TYPE "UDT_DeviceState"
TITLE = UDT_DeviceState
VERSION : 0.1
//User-defined structure of device states.
   STRUCT
      Configure { ExternalAccessible := 'False'; ExternalVisible := 'False'; ExternalWritable := 'False'} : Bool;   // Device configured in TIA Portal hardware
      Exist { ExternalAccessible := 'False'; ExternalVisible := 'False'; ExternalWritable := 'False'} : Bool;   // Device physically connected
      Error { ExternalAccessible := 'False'; ExternalVisible := 'False'; ExternalWritable := 'False'} : Bool;   // Device has an error
      ProfinetNumber : UInt;   // Profinet slave number
      HW_ID : UInt;   // Device's HW_ID
      PNDeviceName : String;   // Device's project name
   END_STRUCT;

END_TYPE

TYPE "UDT_ModuleState"
TITLE = UDT_ModuleState
VERSION : 0.1
//User-defined structure of module states.
   STRUCT
      Configured { ExternalAccessible := 'False'; ExternalVisible := 'False'; ExternalWritable := 'False'} : Bool;   // Module configured
      Exist { ExternalAccessible := 'False'; ExternalVisible := 'False'; ExternalWritable := 'False'} : Bool;   // Module exist
      Error { ExternalAccessible := 'False'; ExternalVisible := 'False'; ExternalWritable := 'False'} : Bool;   // Module has error
   END_STRUCT;

END_TYPE

TYPE "UDT_GINFedEx"
VERSION : 0.1
   STRUCT
      Timestamp : String[17];   // Local time timestamp
      TimeZoneDesignator : String[5];   // Time zone designator
      PackageEntrancePoint : String[14];   // Entrance point, where LLC starts tracking the parcel.
      PackageEntranceState : String[1];   // Entrance state
      PackageExitPoint : String[14];   // Exit point name, where LLC reports the last known tracking point.
      PackageExitState : String[1];   // Exit point state when LLC reports the last known tracking point.
      PalletType : String[2];   // Pallet code for different type of pallets on the market
      Mask : String[1];   // Flag to indicate that a pallet has been mask.
      CellNumber : String[4];   // Tray/Cell number (for loop sorters) or generated by LLC (on line sorters).
      CellsOccupied : String[1];   // Cells occupied by the piece for loop sorters.
      ImageID : String[6];   // Image ID number created by the ADC system.
      ScanUnitType : String[1];   // Scan unit type
      ADCSystemID : String[15];   // Number assigned by the ADC system
      PackageID : String[15];   // Number assigned by the LLC system
      LLCSystemID : String[15];
      HLCPackageID : String[10];   // Unique number for the specific package during it stays in HLC system.
      HLCResultCode : String[16];   // Result code based on processing of the scan event messages.
      ShipmentID : String[6];   // Consignment id of the parcel.
      WeightStatus : String[1];   // Status to indicate if the parcel/pallet has weight on the system.
      ActualDestination : String[6];   // Location code value that describes the actual disposition of the package.
      Destination1 : String[6];   // Location code value that describes where the package should go (Diverter Number).
      Destination2 : String[6];   // Location code value that describes where the package should go (Diverter Number).
      Destination3 : String[6];   // Location code value that describes where the package should go (Diverter Number).
      Destination4 : String[6];   // Location code value that describes where the package should go (Diverter Number).
      Destination5 : String[6];   // Location code value that describes where the package should go (Diverter Number).
      CutOffTimeDestination1 : String[5];   // Cut Off Time in Local Time.
      CutOffTimeDestination2 : String[5];   // Cut Off Time in Local Time.
      CutOffTimeDestination3 : String[5];   // Cut Off Time in Local Time.
      CutOffTimeDestination4 : String[5];   // Cut Off Time in Local Time.
      CutOffTimeDestination5 : String[5];   // Cut Off Time in Local Time.
      ReasonCode1 : String[8];   // Management Code value that describes the result of attempting to route the package to the Destination
      ReasonCode2 : String[8];   // Management Code value that describes the result of attempting to route the package to the Destination
      ReasonCode3 : String[8];   // Management Code value that describes the result of attempting to route the package to the Destination
      ReasonCode4 : String[8];   // Management Code value that describes the result of attempting to route the package to the Destination
      ReasonCode5 : String[8];   // Management Code value that describes the result of attempting to route the package to the Destination
      HLCDataText : String[20];   // Free text for future use.
      Customs : String[1];   // Need to be checked by customs
      DIMSystemID : String[15];   // Identifier of dimensioning system.
      DIMStatus : String[5];   // Basic diagnostic information from the dimensioning system at the moment of the measurement.
      PackageDimLength : String[6];   // Length dimension of package in resolution of dim system.
      PackageDimWidth : String[6];   // Width dimension of package in resolution of dim system.
      PackageDimHeight : String[6];   // Height dimension of package in resolution of dim system.
      DIMUOM : String[2];   // Unit of measure of the package dimensions.
      DimLFTstatusCode : String[8];   // Dimension LFT status code.
      DimConfidence : String[2];   // The level of assurance for the correct dimensions.
      DimensionSource : String[1];   // For combined camera/laser dim acquisition devices. It indicates type of capturing mode
      AlibiDims : String[25];   // Alibi for Dimensions
      SCLSystemID : String[15];   // Identifier of weight scale.
      SCLStatus : String[5];   // Basic diagnostic information from the weight scale system.
      SCLWT : String[6];   // Scale weight of package in resolution of scale system.
      SCLWTUOM : String[2];   // Unit of measurement for Weight
      SCLLFTStatusCode : String[2];   // Scale LFT status code.
      AlibiWeight : String[25];   // Alibi for Weight
      ReasonCode : String[1];   // This code should be used when the SI message has some defect.
      Stackable : String[1];   // If stackable recognition is enabled, Y or N
      Stickerstype : String[2];   // When optical recognition is used to sort
      FlyingDocument : String[1];   // Status to confirm if the document/flyer is prone to fly off the sorter.
      ModeofOperation : String[1];   // Camera Tunnel operational mode format:
      CameraHeadstatus : String[2];   // Diagnostic information on camera/laser heads performing barcode reads.
      PackageDataTruncated : String[1];   // Y = Full length of barcode data exceeds 9999 bytes, data truncated
      TotalBarcodeDataLength : String[4];   // Length of all barcode data that was sent in bytes;
      Barcode1Identification : String[3];   // Barcode identifier code.
      Barcode1status : String[2];   // Barcode confidence factor
      Barcode1datalength : String[4];   // String length of barcode data in bytes; inclusive of this field. Use 0054 as a fixed value
      Barcode1data : String[50];   // Highest priority barcode
      Barcode2Identification : String[3];   // Barcode identifier code.
      Barcode2status : String[2];   // Barcode confidence factor
      Barcode2datalength : String[4];   // String length of barcode data in bytes; inclusive of this field. Use 0054 as a fixed value
      Barcode2data : String[50];   // Highest priority barcode
      Barcode3Identification : String[3];   // Barcode identifier code.
      Barcode3status : String[2];   // Barcode confidence factor
      Barcode3datalength : String[4];   // String length of barcode data in bytes; inclusive of this field. Use 0054 as a fixed value
      Barcode3data : String[50];   // Highest priority barcode
      BarcodeIdentification : String[3];   // Barcode identifier code.
      Barcodestatus : String[2];   // Barcode confidence factor
      Barcodedatalength : String[4];   // String length of barcode data in bytes
      Barcodedata : String[50];   // Sortation barcode
      CustomerID : DInt;   // 6 digits SequentialID (NNNNNN)
      AreaNumber : String[2];   // Package Sequence ID "Area Number"
      PurgeEnabled { ExternalAccessible := 'False'; ExternalVisible := 'False'; ExternalWritable := 'False'} : Bool;   // Purge enabled for parcel: destination overwritten with Purge destination
   END_STRUCT;

END_TYPE

TYPE "UDT_GINStandard"
VERSION : 0.1
   STRUCT
      Destination : Array[0..20] of DInt;   // Destination
      Identification : Struct   // Barcode identification
         GoodRead { ExternalAccessible := 'False'; ExternalVisible := 'False'; ExternalWritable := 'False'} : Bool;   // Barcode read was succesful
         NoRead { ExternalAccessible := 'False'; ExternalVisible := 'False'; ExternalWritable := 'False'} : Bool;   // Barcode read was unsuccesful
         MultiRead { ExternalAccessible := 'False'; ExternalVisible := 'False'; ExternalWritable := 'False'} : Bool;   // Multiple Barcodes were detected
         Barcode : Array[0..10] of Char;   // Barcode values
      END_STRUCT;
      GinAssigned { ExternalAccessible := 'False'; ExternalVisible := 'False'; ExternalWritable := 'False'} : Bool;   // GIN is assigned to package
      Lost { ExternalAccessible := 'False'; ExternalVisible := 'False'; ExternalWritable := 'False'} : Bool;   // Lost in tracking
      Length : Int;   // Length in mm
      Width : Int;   // Width in mm
      Height : Int;   // Height in mm
      Weight : DInt;   // Weight in g
      PkgTooLong { ExternalAccessible := 'False'; ExternalVisible := 'False'; ExternalWritable := 'False'} : Bool;   // Package is too long
      PkgTooSmall { ExternalAccessible := 'False'; ExternalVisible := 'False'; ExternalWritable := 'False'} : Bool;   // Package is too small
      PkgTooHigh { ExternalAccessible := 'False'; ExternalVisible := 'False'; ExternalWritable := 'False'} : Bool;   // Package is too high
      PkgOverWeight { ExternalAccessible := 'False'; ExternalVisible := 'False'; ExternalWritable := 'False'} : Bool;   // Package is over weight
      TrailingGap : Int;   // Trailing gap size in cm between the package
      LeadingGap : Int;   // Leading gap size in cm between the package
      NrOfRecirculations : Int;   // Number of recirculations
      DestReqSend { ExternalAccessible := 'False'; ExternalVisible := 'False'; ExternalWritable := 'False'} : Bool;   // Destination request sent to high level
      DestRcv { ExternalAccessible := 'False'; ExternalVisible := 'False'; ExternalWritable := 'False'} : Bool;   // Destination received from high level
      SortStatus : Struct   // Sort status of the package
         DivertDestination : Int;   // Destination to which the package is diverted
         GoodDivert { ExternalAccessible := 'False'; ExternalVisible := 'False'; ExternalWritable := 'False'} : Bool;   // Package diverted
         FailedDivert { ExternalAccessible := 'False'; ExternalVisible := 'False'; ExternalWritable := 'False'} : Bool;   // Package failed to divert
         NoDivert : Bool := TRUE;   // Divert is not activated
         NoDivertCause : Struct   // Cause for no divert
            ChuteJam { ExternalAccessible := 'False'; ExternalVisible := 'False'; ExternalWritable := 'False'} : Bool;   // Chute is jammed
            ChuteFull { ExternalAccessible := 'False'; ExternalVisible := 'False'; ExternalWritable := 'False'} : Bool;   // Chute is full
            NoRTR { ExternalAccessible := 'False'; ExternalVisible := 'False'; ExternalWritable := 'False'} : Bool;   // Downstream conveyor is not ready to receive
            DestDisabled { ExternalAccessible := 'False'; ExternalVisible := 'False'; ExternalWritable := 'False'} : Bool;   // Destination is disabled
            TrayDisabled { ExternalAccessible := 'False'; ExternalVisible := 'False'; ExternalWritable := 'False'} : Bool;   // Tray is disabled
            SorterNotAtSpeed { ExternalAccessible := 'False'; ExternalVisible := 'False'; ExternalWritable := 'False'} : Bool;   // Sorter is not at speed
            LeadingGapError { ExternalAccessible := 'False'; ExternalVisible := 'False'; ExternalWritable := 'False'} : Bool;   // Gap size with downstream parcel is not enough
            TrailingGapError { ExternalAccessible := 'False'; ExternalVisible := 'False'; ExternalWritable := 'False'} : Bool;   // Gap size with upstream parcel is not enough
            PkgTooHigh { ExternalAccessible := 'False'; ExternalVisible := 'False'; ExternalWritable := 'False'} : Bool;   // Package is too high to divert
            PkgTooLong { ExternalAccessible := 'False'; ExternalVisible := 'False'; ExternalWritable := 'False'} : Bool;   // Package is too long to divert
            DestNotReachable { ExternalAccessible := 'False'; ExternalVisible := 'False'; ExternalWritable := 'False'} : Bool;   // Sort destionation is not reachable
            InvalidDest { ExternalAccessible := 'False'; ExternalVisible := 'False'; ExternalWritable := 'False'} : Bool;   // Sort destination is invalid
            DestTooLate { ExternalAccessible := 'False'; ExternalVisible := 'False'; ExternalWritable := 'False'} : Bool;   // Destination too late
            NoDestRcv { ExternalAccessible := 'False'; ExternalVisible := 'False'; ExternalWritable := 'False'} : Bool;   // Destination not received from high level
         END_STRUCT;
      END_STRUCT;
   END_STRUCT;

END_TYPE

TYPE "UDT_GINWES"
VERSION : 0.1
   STRUCT
      Barcode : String[40];
   END_STRUCT;

END_TYPE

TYPE "UDT_GINWCS"
VERSION : 0.1
   STRUCT
      ActionTaken : String;   // Location code value that describes the actual disposition of the package
      Destination1 : String[20];   // Location code value that describes where the package should go (Diverter Number)
      Destination2 : String[20];   // Location code value that describes where the package should go (Diverter Number)
      Destination3 : String[20];   // Location code value that describes where the package should go (Diverter Number)
      Destination4 : String[20];   // Location code value that describes where the package should go (Diverter Number)
      Destination5 : String[20];   // Location code value that describes where the package should go (Diverter Number)
      ReasonCode : String[2];   // Management Code value that describes the result of attempting to route the package to the Destination
      Barcode1 : String;   // Barcode identifier code
      Barcode2 : String;
      Barcode3 : String;
      Barcode4 : String;
   END_STRUCT;

END_TYPE

TYPE "UDT_GINDHL"
VERSION : 0.1
   STRUCT
      ObjectID : String[10];   // Object ID
      VID : String[16];   // Virtual Item Identifier (VID)
      PieceID : String[40];   // Piece ID barcodes
      SortStrategy : String[1];   // Sort Strategy 1 - Highest priority available , 2 - Nearest
      ParcelReject { ExternalAccessible := 'False'; ExternalVisible := 'False'; ExternalWritable := 'False'} : Bool;   // True - Parcel reject
      Destination : Array[1..6] of Struct   // Destination
         ID : UInt;   // ID
         SortCommandActive { ExternalAccessible := 'False'; ExternalVisible := 'False'; ExternalWritable := 'False'} : Bool;   // Sort command
         ParcelSorted { ExternalAccessible := 'False'; ExternalVisible := 'False'; ExternalWritable := 'False'} : Bool;   // Parcel sorted
         Rejected { ExternalAccessible := 'False'; ExternalVisible := 'False'; ExternalWritable := 'False'} : Bool;   // Parcel rejected
         Reason : Int;   // Reason
      END_STRUCT;
      ParcelLocation : Struct   // Parcel Location
         Current : UInt;   // Current
         Last : UInt;   // Last
         Sort : UInt;   // Sort
      END_STRUCT;
      MFCMessage : Struct   // MFC Sort messages
         Sent : Struct   // Messages sent from the PLC to the MFC system
            SortResult { ExternalAccessible := 'False'; ExternalVisible := 'False'; ExternalWritable := 'False'} : Bool;   // Message Sort Result
            VIDResponse { ExternalAccessible := 'False'; ExternalVisible := 'False'; ExternalWritable := 'False'} : Bool;   // Message VID Response
            ScanReset { ExternalAccessible := 'False'; ExternalVisible := 'False'; ExternalWritable := 'False'} : Bool;   // Message Scan Reset
            XrayResult { ExternalAccessible := 'False'; ExternalVisible := 'False'; ExternalWritable := 'False'} : Bool;   // Message Xray result
            ParcelRegInfo { ExternalAccessible := 'False'; ExternalVisible := 'False'; ExternalWritable := 'False'} : Bool;   // Message Xray registration info
         END_STRUCT;
         Received : Struct   // Messages received from the MFC system to the PLC
            RejectParcel { ExternalAccessible := 'False'; ExternalVisible := 'False'; ExternalWritable := 'False'} : Bool;   // Message Reject Parcel
            Destination { ExternalAccessible := 'False'; ExternalVisible := 'False'; ExternalWritable := 'False'} : Bool;   // Message Destination
            DestinationResent { ExternalAccessible := 'False'; ExternalVisible := 'False'; ExternalWritable := 'False'} : Bool;   // Message Destination Resent
            TemporaryParcelIdentifier { ExternalAccessible := 'False'; ExternalVisible := 'False'; ExternalWritable := 'False'} : Bool;   // Message Temporary Parcel Identifier
            XrayRegistrationInfo { ExternalAccessible := 'False'; ExternalVisible := 'False'; ExternalWritable := 'False'} : Bool;
         END_STRUCT;
      END_STRUCT;
      Xray : Struct   // Xray data structure
         RoutingCode : String[2];   // Routing code
         Group : String[1];   // The group field is used to identify the group of the operator decisions came from in a
         Level : String[1];   // Level field is used to identify which level the operator decision came from in a
         Result : String[1];   // Results can be indicated with the following:A = Accept, R = Reject, U = Unavailable (Timeout), Z = High Threat
         BagIDMessage : Struct   // Message from PLC to Xray
            MessagePrepared { ExternalAccessible := 'False'; ExternalVisible := 'False'; ExternalWritable := 'False'} : Bool;   // The message is prepared and ready to send
            WrongMessageStructure { ExternalAccessible := 'False'; ExternalVisible := 'False'; ExternalWritable := 'False'} : Bool;   // The message has wrong structure
            Sent { ExternalAccessible := 'False'; ExternalVisible := 'False'; ExternalWritable := 'False'} : Bool;   // The message sent by PLC to Xray
            SentTime : String;   // Time when message sent by PLC to Xray
            NotSent { ExternalAccessible := 'False'; ExternalVisible := 'False'; ExternalWritable := 'False'} : Bool;   // The message was not sent from the PLC
            Received { ExternalAccessible := 'False'; ExternalVisible := 'False'; ExternalWritable := 'False'} : Bool;   // The message received by Xray
            TimeReceived : String;   // Time when message received by Xray
            NotReceived { ExternalAccessible := 'False'; ExternalVisible := 'False'; ExternalWritable := 'False'} : Bool;   // The message did not reach Xray
         END_STRUCT;
         DecisionMessage : Struct   // Message from Xray to PLC
            Received { ExternalAccessible := 'False'; ExternalVisible := 'False'; ExternalWritable := 'False'} : Bool;   // The message received by PLC
            ReceivedTime : String;   // The message received by PLC
            NotReceivedOnTime { ExternalAccessible := 'False'; ExternalVisible := 'False'; ExternalWritable := 'False'} : Bool;   // The message did not reach PLC
         END_STRUCT;
      END_STRUCT;
   END_STRUCT;

END_TYPE

TYPE "UDT_CommonStatus"
TITLE = UDT_CommonStatus
VERSION : 0.1
//User-defined structure of common statuses.
   STRUCT
      SafetyStop { ExternalAccessible := 'False'; ExternalVisible := 'False'; ExternalWritable := 'False'} : Bool;   // Emergancy stop
      Error { ExternalAccessible := 'False'; ExternalVisible := 'False'; ExternalWritable := 'False'} : Bool;   // An error is active
      Warning { ExternalAccessible := 'False'; ExternalVisible := 'False'; ExternalWritable := 'False'} : Bool;   // A warning is active
      ManualRun { ExternalAccessible := 'False'; ExternalVisible := 'False'; ExternalWritable := 'False'} : Bool;   // Running in manual mode
      Manual { ExternalAccessible := 'False'; ExternalVisible := 'False'; ExternalWritable := 'False'} : Bool;   // In manual mode
      Halted { ExternalAccessible := 'False'; ExternalVisible := 'False'; ExternalWritable := 'False'} : Bool;   // Halted
      Dieback { ExternalAccessible := 'False'; ExternalVisible := 'False'; ExternalWritable := 'False'} : Bool;   // In dieback
      Stopped { ExternalAccessible := 'False'; ExternalVisible := 'False'; ExternalWritable := 'False'} : Bool;   // Stopped
      Running { ExternalAccessible := 'False'; ExternalVisible := 'False'; ExternalWritable := 'False'} : Bool;   // Running
      EnergySave { ExternalAccessible := 'False'; ExternalVisible := 'False'; ExternalWritable := 'False'} : Bool;   // In energy saving mode
      AutoON { ExternalAccessible := 'False'; ExternalVisible := 'False'; ExternalWritable := 'False'} : Bool;   // Automatic started
   END_STRUCT;

END_TYPE

TYPE "UDT_EventStatistic"
TITLE = UDT_EventStatistic
VERSION : 0.1
//User-defined structure of event statistic data.
   STRUCT
      NumberOfTimes : DInt;   // Number of times the event occurred since last reset
      LastEventSeconds : DInt;   // Number of seconds of the current or last event
      TotalEventSeconds : DInt;   // Total number of seconds the event occurred since last reset
   END_STRUCT;

END_TYPE

TYPE "UDT_GINUPS"
VERSION : 0.1
   STRUCT
      TRKNUM : String[18];   // Tracking number
      PKGUID : String[32];   // Package ID
      MSGID : String[32];   // Message ID
      Length : Int;   // Camera Length in mm
      Width : Int;   // Camera Width in mm
      Height : Int;   // Camera Height in mm
      Weight : DInt;   // Weight in g
      IDCreated { ExternalAccessible := 'False'; ExternalVisible := 'False'; ExternalWritable := 'False'} : Bool;   // Byte 1, Bit 0 - PLCID created or TrayID Read
      DimDataRcv { ExternalAccessible := 'False'; ExternalVisible := 'False'; ExternalWritable := 'False'} : Bool;   // Byte 1, Bit 1 - Package Dimensional Data Received via Camera Scan Data Message
      PkgWrongInduct { ExternalAccessible := 'False'; ExternalVisible := 'False'; ExternalWritable := 'False'} : Bool;   // Byte 1, Bit 2 - Package Did NOT Induct Properly (Non-Tray Systems)
      IDCalcFromCamID { ExternalAccessible := 'False'; ExternalVisible := 'False'; ExternalWritable := 'False'} : Bool;   // Byte 2, Bit 0 - PLCID/TrayID Calculated From CamID
      UnknownParcelID { ExternalAccessible := 'False'; ExternalVisible := 'False'; ExternalWritable := 'False'} : Bool;   // Byte 2, Bit 4 - Unknown Parcel ID
      UndefinedProblem { ExternalAccessible := 'False'; ExternalVisible := 'False'; ExternalWritable := 'False'} : Bool;   // Byte 2, Bit 5 - Un-Defined Problem
      UnrecognizedCmd { ExternalAccessible := 'False'; ExternalVisible := 'False'; ExternalWritable := 'False'} : Bool;   // Byte 2, Bit 6 - Un-recognized command
      SorterInMainteneceMode { ExternalAccessible := 'False'; ExternalVisible := 'False'; ExternalWritable := 'False'} : Bool;   // Byte 2, Bit 7 - Sorter in Maintenance/Commissioning Mode
      DestUserSusp { ExternalAccessible := 'False'; ExternalVisible := 'False'; ExternalWritable := 'False'} : Bool;   // Byte 3, Bit 3 - Destination User Suspended
      SorterNotSynch { ExternalAccessible := 'False'; ExternalVisible := 'False'; ExternalWritable := 'False'} : Bool;   // Byte 3, Bit 6 - Sorter NOT Synchronized (Tilt Tray Systems)
      PkgDetAtVerCheckPoint { ExternalAccessible := 'False'; ExternalVisible := 'False'; ExternalWritable := 'False'} : Bool;   // Byte 4, Bit 0 - Package Detected at Verification Check Point
      ChuteFullAftrAlterDest { ExternalAccessible := 'False'; ExternalVisible := 'False'; ExternalWritable := 'False'} : Bool;   // Byte 4, Bit 7 - Preferred chute full after passed alternate destination
      ChuteNotAvailAfterAlterDest { ExternalAccessible := 'False'; ExternalVisible := 'False'; ExternalWritable := 'False'} : Bool;   // Byte 5, Bit 0 - Preferred chute not available after passed alternate destination
      PLCRedirected { ExternalAccessible := 'False'; ExternalVisible := 'False'; ExternalWritable := 'False'} : Bool;   // Byte 5, Bit 2 - PLC Redirected
      ThreatParcel { ExternalAccessible := 'False'; ExternalVisible := 'False'; ExternalWritable := 'False'} : Bool;   // Threat parcel
   END_STRUCT;

END_TYPE

TYPE "UDT_ProfinetDevice"
TITLE = UDT_ProfinetDevice
VERSION : 0.1
//User-defined structure of profinet device state.
   STRUCT
      DeviceState : "UDT_DeviceState";   // Device state
      Module { S7_SetPoint := 'False'} : Array[0..31] of "UDT_ModuleState";   // Modules
   END_STRUCT;

END_TYPE

TYPE "UDT_Message"
TITLE = UDT_Message
VERSION : 0.1
//User-defined structure of the message characters array.
   STRUCT
      Character : Array[0..499] of Char;   // Message character
   END_STRUCT;

END_TYPE

TYPE "UDT_FifoHeader"
TITLE = UDT_FifoHeader
VERSION : 0.1
//User-defined structure of FIFO register header information.
   STRUCT
      Status : Struct   // Status bits
         Empty { ExternalAccessible := 'False'; ExternalVisible := 'False'; ExternalWritable := 'False'} : Bool;   // FIFO Empty
         Prefull { ExternalAccessible := 'False'; ExternalVisible := 'False'; ExternalWritable := 'False'} : Bool;   // FIFO Prefull
         Full { ExternalAccessible := 'False'; ExternalVisible := 'False'; ExternalWritable := 'False'} : Bool;   // FIFO Full
      END_STRUCT;
      NextEntryToRead : Int;   // Next FIFO entry to read
      NextEntryToWrite : Int;   // Next FIFO entry to write
      MaxNrOfEntries : Int;   // Maximum number of FIFO entries
      TotalEntriesStored : Int;   // Total number of FIFO entries
   END_STRUCT;

END_TYPE

TYPE "UDT_ProfiDiagStatistics"
TITLE = UDT_ProfiDiagStatistics
VERSION : 0.1
//User-defined structure of FB_ProfiDiag function block statistics.
   STRUCT
      DeviceError { S7_SetPoint := 'False'} : Array[0..512] of "UDT_EventStatistic";   // Device error statistics
   END_STRUCT;

END_TYPE

TYPE "UDT_Connection"
TITLE = UDT_Connection
VERSION : 0.1
//User-defined structure of connection parameters.
   STRUCT
      ActiveEstablished : Bool := FALSE;   // 0 – Passive connection establishment; 1 – Active connection establishment
      Interface_ID : HW_ANY := 64;   // Interface ID of CPU Ethernet interface
      ID : CONN_OUC;   // Unique ID as system reference for the connection
      IP : Array[1..4] of Int;   // IP address
      Port : UInt;   // Port number of the communication partner
      ConTimeout : DInt;   // Maximum waiting time for response from the communication partner [ms]
   END_STRUCT;

END_TYPE

TYPE "UDT_PowerDistributionPanelCBState"
VERSION : 0.1
   STRUCT
      CircuitBreakerStateF100 { ExternalAccessible := 'False'; ExternalVisible := 'False'; ExternalWritable := 'False'} : Bool;   // Circuit Breaker State Ok if the signal is true
      CircuitBreakerStateF201 { ExternalAccessible := 'False'; ExternalVisible := 'False'; ExternalWritable := 'False'} : Bool;   // Circuit Breaker State Ok if the signal is true
      CircuitBreakerStateF202 { ExternalAccessible := 'False'; ExternalVisible := 'False'; ExternalWritable := 'False'} : Bool;   // Circuit Breaker State Ok if the signal is true
      CircuitBreakerStateF203 { ExternalAccessible := 'False'; ExternalVisible := 'False'; ExternalWritable := 'False'} : Bool;   // Circuit Breaker State Ok if the signal is true
      CircuitBreakerStateF204 { ExternalAccessible := 'False'; ExternalVisible := 'False'; ExternalWritable := 'False'} : Bool;   // Circuit Breaker State Ok if the signal is true
      CircuitBreakerStateF205 { ExternalAccessible := 'False'; ExternalVisible := 'False'; ExternalWritable := 'False'} : Bool;   // Circuit Breaker State Ok if the signal is true
      CircuitBreakerStateF206 { ExternalAccessible := 'False'; ExternalVisible := 'False'; ExternalWritable := 'False'} : Bool;   // Circuit Breaker State Ok if the signal is true
      CircuitBreakerStateF207 { ExternalAccessible := 'False'; ExternalVisible := 'False'; ExternalWritable := 'False'} : Bool;   // Circuit Breaker State Ok if the signal is true
      CircuitBreakerStateF208 { ExternalAccessible := 'False'; ExternalVisible := 'False'; ExternalWritable := 'False'} : Bool;   // Circuit Breaker State Ok if the signal is true
      CircuitBreakerStateF209 { ExternalAccessible := 'False'; ExternalVisible := 'False'; ExternalWritable := 'False'} : Bool;   // Circuit Breaker State Ok if the signal is true
      CircuitBreakerStateF210 { ExternalAccessible := 'False'; ExternalVisible := 'False'; ExternalWritable := 'False'} : Bool;   // Circuit Breaker State Ok if the signal is true
      CircuitBreakerStateF211 { ExternalAccessible := 'False'; ExternalVisible := 'False'; ExternalWritable := 'False'} : Bool;   // Circuit Breaker State Ok if the signal is true
      CircuitBreakerStateF212 { ExternalAccessible := 'False'; ExternalVisible := 'False'; ExternalWritable := 'False'} : Bool;   // Circuit Breaker State Ok if the signal is true
      CircuitBreakerStateF213 { ExternalAccessible := 'False'; ExternalVisible := 'False'; ExternalWritable := 'False'} : Bool;   // Circuit Breaker State Ok if the signal is true
      CircuitBreakerStateF214 { ExternalAccessible := 'False'; ExternalVisible := 'False'; ExternalWritable := 'False'} : Bool;   // Circuit Breaker State Ok if the signal is true
      CircuitBreakerStateF215 { ExternalAccessible := 'False'; ExternalVisible := 'False'; ExternalWritable := 'False'} : Bool;   // Circuit Breaker State Ok if the signal is true
      CircuitBreakerStateF216 { ExternalAccessible := 'False'; ExternalVisible := 'False'; ExternalWritable := 'False'} : Bool;   // Circuit Breaker State Ok if the signal is true
      CircuitBreakerStateF217 { ExternalAccessible := 'False'; ExternalVisible := 'False'; ExternalWritable := 'False'} : Bool;   // Circuit Breaker State Ok if the signal is true
      CircuitBreakerStateF218 { ExternalAccessible := 'False'; ExternalVisible := 'False'; ExternalWritable := 'False'} : Bool;   // Circuit Breaker State Ok if the signal is true
      CircuitBreakerStateF219 { ExternalAccessible := 'False'; ExternalVisible := 'False'; ExternalWritable := 'False'} : Bool;   // Circuit Breaker State Ok if the signal is true
      CircuitBreakerStateF220 { ExternalAccessible := 'False'; ExternalVisible := 'False'; ExternalWritable := 'False'} : Bool;   // Circuit Breaker State Ok if the signal is true
      CircuitBreakerStateF221 { ExternalAccessible := 'False'; ExternalVisible := 'False'; ExternalWritable := 'False'} : Bool;   // Circuit Breaker State Ok if the signal is true
      CircuitBreakerStateF222 { ExternalAccessible := 'False'; ExternalVisible := 'False'; ExternalWritable := 'False'} : Bool;   // Circuit Breaker State Ok if the signal is true
      CircuitBreakerStateF223 { ExternalAccessible := 'False'; ExternalVisible := 'False'; ExternalWritable := 'False'} : Bool;   // Circuit Breaker State Ok if the signal is true
      CircuitBreakerStateF224 { ExternalAccessible := 'False'; ExternalVisible := 'False'; ExternalWritable := 'False'} : Bool;   // Circuit Breaker State Ok if the signal is true
      CircuitBreakerStateF225 { ExternalAccessible := 'False'; ExternalVisible := 'False'; ExternalWritable := 'False'} : Bool;   // Circuit Breaker State Ok if the signal is true
      CircuitBreakerStateF226 { ExternalAccessible := 'False'; ExternalVisible := 'False'; ExternalWritable := 'False'} : Bool;   // Circuit Breaker State Ok if the signal is true
      CircuitBreakerStateF227 { ExternalAccessible := 'False'; ExternalVisible := 'False'; ExternalWritable := 'False'} : Bool;   // Circuit Breaker State Ok if the signal is true
      CircuitBreakerStateF228 { ExternalAccessible := 'False'; ExternalVisible := 'False'; ExternalWritable := 'False'} : Bool;   // Circuit Breaker State Ok if the signal is true
      CircuitBreakerStateF229 { ExternalAccessible := 'False'; ExternalVisible := 'False'; ExternalWritable := 'False'} : Bool;   // Circuit Breaker State Ok if the signal is true
      CircuitBreakerStateF230 { ExternalAccessible := 'False'; ExternalVisible := 'False'; ExternalWritable := 'False'} : Bool;   // Circuit Breaker State Ok if the signal is true
      CircuitBreakerStateF231 { ExternalAccessible := 'False'; ExternalVisible := 'False'; ExternalWritable := 'False'} : Bool;   // Circuit Breaker State Ok if the signal is true
      CircuitBreakerStateF232 { ExternalAccessible := 'False'; ExternalVisible := 'False'; ExternalWritable := 'False'} : Bool;   // Circuit Breaker State Ok if the signal is true
      CircuitBreakerStateF233 { ExternalAccessible := 'False'; ExternalVisible := 'False'; ExternalWritable := 'False'} : Bool;   // Circuit Breaker State Ok if the signal is true
      CircuitBreakerStateF234 { ExternalAccessible := 'False'; ExternalVisible := 'False'; ExternalWritable := 'False'} : Bool;   // Circuit Breaker State Ok if the signal is true
      CircuitBreakerStateF235 { ExternalAccessible := 'False'; ExternalVisible := 'False'; ExternalWritable := 'False'} : Bool;   // Circuit Breaker State Ok if the signal is true
      CircuitBreakerStateF236 { ExternalAccessible := 'False'; ExternalVisible := 'False'; ExternalWritable := 'False'} : Bool;   // Circuit Breaker State Ok if the signal is true
      CircuitBreakerStateF237 { ExternalAccessible := 'False'; ExternalVisible := 'False'; ExternalWritable := 'False'} : Bool;   // Circuit Breaker State Ok if the signal is true
      CircuitBreakerStateF238 { ExternalAccessible := 'False'; ExternalVisible := 'False'; ExternalWritable := 'False'} : Bool;   // Circuit Breaker State Ok if the signal is true
      CircuitBreakerStateF239 { ExternalAccessible := 'False'; ExternalVisible := 'False'; ExternalWritable := 'False'} : Bool;   // Circuit Breaker State Ok if the signal is true
      CircuitBreakerStateF240 { ExternalAccessible := 'False'; ExternalVisible := 'False'; ExternalWritable := 'False'} : Bool;   // Circuit Breaker State Ok if the signal is true
      CircuitBreakerStateF241 { ExternalAccessible := 'False'; ExternalVisible := 'False'; ExternalWritable := 'False'} : Bool;   // Circuit Breaker State Ok if the signal is true
      CircuitBreakerStateF242 { ExternalAccessible := 'False'; ExternalVisible := 'False'; ExternalWritable := 'False'} : Bool;   // Circuit Breaker State Ok if the signal is true
      CircuitBreakerStateF243 { ExternalAccessible := 'False'; ExternalVisible := 'False'; ExternalWritable := 'False'} : Bool;   // Circuit Breaker State Ok if the signal is true
      CircuitBreakerStateF244 { ExternalAccessible := 'False'; ExternalVisible := 'False'; ExternalWritable := 'False'} : Bool;   // Circuit Breaker State Ok if the signal is true
      CircuitBreakerStateF245 { ExternalAccessible := 'False'; ExternalVisible := 'False'; ExternalWritable := 'False'} : Bool;   // Circuit Breaker State Ok if the signal is true
      CircuitBreakerStateF246 { ExternalAccessible := 'False'; ExternalVisible := 'False'; ExternalWritable := 'False'} : Bool;   // Circuit Breaker State Ok if the signal is true
      CircuitBreakerStateF247 { ExternalAccessible := 'False'; ExternalVisible := 'False'; ExternalWritable := 'False'} : Bool;   // Circuit Breaker State Ok if the signal is true
      CircuitBreakerStateF248 { ExternalAccessible := 'False'; ExternalVisible := 'False'; ExternalWritable := 'False'} : Bool;   // Circuit Breaker State Ok if the signal is true
      CircuitBreakerStateF249 { ExternalAccessible := 'False'; ExternalVisible := 'False'; ExternalWritable := 'False'} : Bool;   // Circuit Breaker State Ok if the signal is true
      CircuitBreakerStateF250 { ExternalAccessible := 'False'; ExternalVisible := 'False'; ExternalWritable := 'False'} : Bool;   // Circuit Breaker State Ok if the signal is true
      CircuitBreakerStateF251 { ExternalAccessible := 'False'; ExternalVisible := 'False'; ExternalWritable := 'False'} : Bool;   // Circuit Breaker State Ok if the signal is true
      CircuitBreakerStateF501 { ExternalAccessible := 'False'; ExternalVisible := 'False'; ExternalWritable := 'False'} : Bool;   // Circuit Breaker State Ok if the signal is true
      CircuitBreakerStateF502 { ExternalAccessible := 'False'; ExternalVisible := 'False'; ExternalWritable := 'False'} : Bool;   // Circuit Breaker State Ok if the signal is true
      CircuitBreakerStateF503 { ExternalAccessible := 'False'; ExternalVisible := 'False'; ExternalWritable := 'False'} : Bool;   // Circuit Breaker State Ok if the signal is true
      CircuitBreakerStateF504 { ExternalAccessible := 'False'; ExternalVisible := 'False'; ExternalWritable := 'False'} : Bool;   // Circuit Breaker State Ok if the signal is true
      CircuitBreakerStateF505 { ExternalAccessible := 'False'; ExternalVisible := 'False'; ExternalWritable := 'False'} : Bool;   // Circuit Breaker State Ok if the signal is true
   END_STRUCT;

END_TYPE

TYPE "UDT_EquipmentControl"
TITLE = UDT_EquipmentControl
VERSION : 0.1
//User-defined structure of equipment control commands.
   STRUCT
      Command : Struct   // Control command
         Start { ExternalAccessible := 'False'; ExternalVisible := 'False'; ExternalWritable := 'False'} : Bool;   // Start conveyor
         Stop { ExternalAccessible := 'False'; ExternalVisible := 'False'; ExternalWritable := 'False'} : Bool;   // Stop conveyor
         Reset { ExternalAccessible := 'False'; ExternalVisible := 'False'; ExternalWritable := 'False'} : Bool;   // Faults reset
         ResetData { ExternalAccessible := 'False'; ExternalVisible := 'False'; ExternalWritable := 'False'} : Bool;   // Statistics reset
         ManualMode { ExternalAccessible := 'False'; ExternalVisible := 'False'; ExternalWritable := 'False'} : Bool;   // Manual mode required
         DisableManualMode { ExternalAccessible := 'False'; ExternalVisible := 'False'; ExternalWritable := 'False'} : Bool;   // Disable manual mode
         AutomaticOn { ExternalAccessible := 'False'; ExternalVisible := 'False'; ExternalWritable := 'False'} : Bool;   // System is started in automatic mode
         StopRequest { ExternalAccessible := 'False'; ExternalVisible := 'False'; ExternalWritable := 'False'} : Bool;
      END_STRUCT;
      Report { S7_SetPoint := 'False'} : "UDT_CommonStatus";   // Conveyors state
      Request : Struct   // Request from equipment
         RestartRequired { ExternalAccessible := 'False'; ExternalVisible := 'False'; ExternalWritable := 'False'} : Bool;   // Restart required from system control
         SignalingRequest { ExternalAccessible := 'False'; ExternalVisible := 'False'; ExternalWritable := 'False'} : Bool;   // Beeper required
         InhibitStop { ExternalAccessible := 'False'; ExternalVisible := 'False'; ExternalWritable := 'False'} : Bool;
      END_STRUCT;
   END_STRUCT;

END_TYPE

TYPE "UDT_ProfinetNetwork"
TITLE = UDT_ProfinetNetwork
VERSION : 0.1
//User-defined structure of profinet network state.
   STRUCT
      DeviceStatus : Array[0..512] of "UDT_ProfinetDevice";   // Profinet device status
   END_STRUCT;

END_TYPE

TYPE "UDT_ControlPowerGroupStatistics"
VERSION : 0.1
   STRUCT
      PowerSupplyGroupWarnning : "UDT_EventStatistic";   // Warning Power Supply Group Statistics
      PowerSupplyGroupError : "UDT_EventStatistic";   // Error Power Supply Group Statistics
   END_STRUCT;

END_TYPE

TYPE "UDT_TCPIPConnectStatistics"
TITLE = UDT_TCPIPConnectStatistics
VERSION : 0.1
//User-defined structure of FB_TCPIPConnect function block statistics.
   STRUCT
      ConnectionLost { S7_SetPoint := 'False'} : "UDT_EventStatistic";   // Connection lost statistics
   END_STRUCT;

END_TYPE

TYPE "UDT_TCPIPReceiveStatistics"
TITLE = UDT_TCPIPReceiveStatistics
VERSION : 0.1
//User-defined structure of FB_TCPIPReceive function block statistics.
   STRUCT
      InvalidMsg : UInt;   // Invalid message received
   END_STRUCT;

END_TYPE

TYPE "UDT_WSRBufferState"
VERSION : 0.1
   STRUCT
      Destination : Int;
      BufferState1 : Struct
         BinRequest : Bool;
         BinSend : Bool;
         UpcomingBarcode : String[30];
         WaintingTime : Int;
      END_STRUCT;
      BufferState2 : Struct
         BinRequest : Bool;
         BinSend : Bool;
         UpcomingBarcode : String[30];
         WaintingTime : Int;
      END_STRUCT;
      BufferState3 : Struct
         BinRequest : Bool;
         BinSend : Bool;
         UpcomingBarcode : String[30];
         WaintingTime : Int;
      END_STRUCT;
   END_STRUCT;

END_TYPE

TYPE "UDT_SystemControlStatus"
TITLE = UDT_SystemControlStatus
VERSION : 0.1
//User-defined structure of FB_SystemControl function block status.
   STRUCT
      Status : Int;   // Status number
   END_STRUCT;

END_TYPE

TYPE "UDT_ControlPowerGroupStatus"
VERSION : 0.1
   STRUCT
      Status : Int;   // Status number
      Specific : Struct
         Fail_PowerSupply_1 { ExternalAccessible := 'False'; ExternalVisible := 'False'; ExternalWritable := 'False'} : Bool;   // Power supply 1 fail
         Fail_PowerSupply_2 { ExternalAccessible := 'False'; ExternalVisible := 'False'; ExternalWritable := 'False'} : Bool;   // Power supply 2 fail
         Fail_PowerSupply_3 { ExternalAccessible := 'False'; ExternalVisible := 'False'; ExternalWritable := 'False'} : Bool;   // Power supply 3 fail
         Fail_PowerSupply_4 { ExternalAccessible := 'False'; ExternalVisible := 'False'; ExternalWritable := 'False'} : Bool;   // Power supply 4 fail
         Fail_PowerSupply_5 { ExternalAccessible := 'False'; ExternalVisible := 'False'; ExternalWritable := 'False'} : Bool;   // Power supply 5 fail
         Fail_PowerSupply_6 { ExternalAccessible := 'False'; ExternalVisible := 'False'; ExternalWritable := 'False'} : Bool;   // Power supply 6 fail
         Fail_PowerSupply_7 { ExternalAccessible := 'False'; ExternalVisible := 'False'; ExternalWritable := 'False'} : Bool;   // Power supply 7 fail
         Fail_PowerSupply_8 { ExternalAccessible := 'False'; ExternalVisible := 'False'; ExternalWritable := 'False'} : Bool;   // Power supply 8 fail
         Fail_PowerSupply_9 { ExternalAccessible := 'False'; ExternalVisible := 'False'; ExternalWritable := 'False'} : Bool;   // Power supply 9 fail
         Fail_PowerSupply_10 { ExternalAccessible := 'False'; ExternalVisible := 'False'; ExternalWritable := 'False'} : Bool;   // Power supply 10 fail
         PowerSuppliesWarning { ExternalAccessible := 'False'; ExternalVisible := 'False'; ExternalWritable := 'False'} : Bool;   // Power supplies warning
         PowerSuppliesError { ExternalAccessible := 'False'; ExternalVisible := 'False'; ExternalWritable := 'False'} : Bool;   // Power supplies error
      END_STRUCT;
   END_STRUCT;

END_TYPE

TYPE "UDT_MainControlPanelStatus"
TITLE = Cabinet MCP Status
VERSION : 0.1
   STRUCT
      Status : Int;   //  Status number
      Specific : Struct
         PN_PN_MSP_PNSlaveNotOnline { ExternalAccessible := 'False'; ExternalVisible := 'False'; ExternalWritable := 'False'} : Bool;   //  PNPN coupler is not online
         PN_PN_MSP_PNSlaveError { ExternalAccessible := 'False'; ExternalVisible := 'False'; ExternalWritable := 'False'} : Bool;   //  PNPN coupler has an error
         PN_PN_MSP_PNSlaveWarning { ExternalAccessible := 'False'; ExternalVisible := 'False'; ExternalWritable := 'False'} : Bool;   //  PNPN coupler has a warning
         IOModule_PNSlaveNotOnline { ExternalAccessible := 'False'; ExternalVisible := 'False'; ExternalWritable := 'False'} : Bool;   // I/O Module is not online
         IOModule_PNSlaveError { ExternalAccessible := 'False'; ExternalVisible := 'False'; ExternalWritable := 'False'} : Bool;   // I/O Module has an error
         IOModule_PNSlaveWarning { ExternalAccessible := 'False'; ExternalVisible := 'False'; ExternalWritable := 'False'} : Bool;   // I/O Module has a warning
         ScalanceSwitchPNSlaveNotOnline { ExternalAccessible := 'False'; ExternalVisible := 'False'; ExternalWritable := 'False'} : Bool;   // Scalance switch is not online
         ScalanceSwitchPNSlaveError { ExternalAccessible := 'False'; ExternalVisible := 'False'; ExternalWritable := 'False'} : Bool;   // Scalance switch has an error
         ScalanceSwitchPNSlaveWarning { ExternalAccessible := 'False'; ExternalVisible := 'False'; ExternalWritable := 'False'} : Bool;   // Scalance switch has a warning
         ScalanceSwitchStatus { ExternalAccessible := 'False'; ExternalVisible := 'False'; ExternalWritable := 'False'} : Bool;   // TRUE when Scalance switch is not healthy
         Singulator_PNSlaveNotOnline { ExternalAccessible := 'False'; ExternalVisible := 'False'; ExternalWritable := 'False'} : Bool;   // Singulator coupler is not online
         Singulator_PNSlaveError { ExternalAccessible := 'False'; ExternalVisible := 'False'; ExternalWritable := 'False'} : Bool;   // Singulator coupler has an error
         Singulator_PNSlaveWarning { ExternalAccessible := 'False'; ExternalVisible := 'False'; ExternalWritable := 'False'} : Bool;   // Singulator coupler has a warning
         UPSSwitchTripped { ExternalAccessible := 'False'; ExternalVisible := 'False'; ExternalWritable := 'False'} : Bool;   //  Unit Power Supply switch tripped
         FireAlarmActive { ExternalAccessible := 'False'; ExternalVisible := 'False'; ExternalWritable := 'False'} : Bool;   //  Fire alarm active when the signal is true
         PS_201T1_Tripped { ExternalAccessible := 'False'; ExternalVisible := 'False'; ExternalWritable := 'False'} : Bool;   //  TRUE if power supply 201T1 tripped
         "230VAC_CB201F4Tripped" { ExternalAccessible := 'False'; ExternalVisible := 'False'; ExternalWritable := 'False'} : Bool;   //  TRUE if MCP circuit breaker 201F4 tripped
         "230VAC_CB101F1Tripped" { ExternalAccessible := 'False'; ExternalVisible := 'False'; ExternalWritable := 'False'} : Bool;   //  TRUE if MCP circuit breaker 101F1 tripped
         "230VAC_CB101F4Tripped" { ExternalAccessible := 'False'; ExternalVisible := 'False'; ExternalWritable := 'False'} : Bool;   //  TRUE if MCP circuit breaker 101F4 tripped
         "230VAC_CB102F1Tripped" { ExternalAccessible := 'False'; ExternalVisible := 'False'; ExternalWritable := 'False'} : Bool;   //  TRUE if MCU circuit breaker 102F1 tripped
         "230VAC_CB102F3Tripped" { ExternalAccessible := 'False'; ExternalVisible := 'False'; ExternalWritable := 'False'} : Bool;   //  TRUE if MCU circuit breaker 102F3 tripped
         "24VDC_CB201F1Tripped" { ExternalAccessible := 'False'; ExternalVisible := 'False'; ExternalWritable := 'False'} : Bool;   //  TRUE if MCU circuit breaker 205F1 tripped
         "24VDC_CB205F5Tripped" { ExternalAccessible := 'False'; ExternalVisible := 'False'; ExternalWritable := 'False'} : Bool;   //  TRUE if MCU circuit breaker 205F5 tripped
         "24VDC_CB205F9Tripped" { ExternalAccessible := 'False'; ExternalVisible := 'False'; ExternalWritable := 'False'} : Bool;   //  TRUE if MCU circuit breaker 205F9 tripped
         Spare_1 { ExternalAccessible := 'False'; ExternalVisible := 'False'; ExternalWritable := 'False'} : Bool;   // Spare
         Spare_2 { ExternalAccessible := 'False'; ExternalVisible := 'False'; ExternalWritable := 'False'} : Bool;   // Spare
         Spare_3 { ExternalAccessible := 'False'; ExternalVisible := 'False'; ExternalWritable := 'False'} : Bool;   // Spare
         RackSlotError : Array[0..31] of Bool;   //  One of the main rack slots has an error
         IOModuleSlotError : Array[0..31] of Bool;   //  Module error
      END_STRUCT;
   END_STRUCT;

END_TYPE

TYPE "UDT_TCPIPConnectStatus"
TITLE = UDT_TCPIPConnectStatus
VERSION : 0.1
//User-defined structure of FB_TCPIPConnect function block status.
   STRUCT
      Status : Int;   // Status number
      Specific : Struct   // Specific status structure
         ErrorCode : Struct   // Error code structure
            TCON : Word;   // Siemens TCON error code - Check documetation
            TDISCON : Word;   // Siemens TDISCON error code - Check documetation
            TDIAG : Word;   // Siemens TDIAG error code - Check documetation
         END_STRUCT;
         Connected { ExternalAccessible := 'False'; ExternalVisible := 'False'; ExternalWritable := 'False'} : Bool;   // Connected
         CommunicationFault { ExternalAccessible := 'False'; ExternalVisible := 'False'; ExternalWritable := 'False'} : Bool;   // Communication fault
      END_STRUCT;
   END_STRUCT;

END_TYPE

TYPE "UDT_UnknownGIN"
TITLE = UDT_UnknownGIN
VERSION : 0.1
//User-defined structure of unknown GIN range.
   STRUCT
      Start : Int := 1;   // Unknown GIN range start value
      End : Int := 199;   // Unknown GIN range end value
      GIN : Int := 0;   // Las generated unknown GIN
   END_STRUCT;

END_TYPE

TYPE "UDT_GOSLog"
VERSION : 0.1
   STRUCT
      GIN_nr : Int;
      InfeedUpstreamGap : Int;   // Gap in millimeters (mm)
      InfeedDownstreamGap : Int;   // Gap in millimeters (mm)
      OutfeedUpstreamGap : Int;   // Gap in meters (mm)
      OutfeedDownstreamGap : Int;   // Gap in meters (mm)
      ParcelLength : Int;
      GapToBeRecovered : Int;
      ParcelDownStreamResults : Int;
      ParcelUpStreamResults : Int;
      Accelerate { ExternalAccessible := 'False'; ExternalVisible := 'False'; ExternalWritable := 'False'} : Bool;
      Decelerate { ExternalAccessible := 'False'; ExternalVisible := 'False'; ExternalWritable := 'False'} : Bool;
      PrevConveyorUpstreamGap : Int;
      PrevConveyorDownstreamGap : Int;
      NextConveyorUpstreamGap : Int;
      NextConveyorDownstreamGap : Int;
   END_STRUCT;

END_TYPE

TYPE "UDT_GIN"
VERSION : 0.1
   STRUCT
      General { S7_SetPoint := 'False'} : "UDT_GINStandard";
      FedEx { S7_SetPoint := 'False'} : "UDT_GINFedEx";
      UPS { S7_SetPoint := 'False'} : "UDT_GINUPS";
      DHL { S7_SetPoint := 'False'} : "UDT_GINDHL";
      WCS { S7_SetPoint := 'False'} : "UDT_GINWCS";
      WES { S7_SetPoint := 'False'} : "UDT_GINWES";
   END_STRUCT;

END_TYPE

TYPE "UDT_MainControlPanelStatistics"
TITLE = Cabinet MCP Statistics
VERSION : 0.1
   STRUCT
      UPSFault : "UDT_EventStatistic";   // Unit Power Supply fault statistics
      FireAlarm : "UDT_EventStatistic";   // Fire Alarm active statistics
      "230VAC_CB101F1Tripped" : "UDT_EventStatistic";   // Circuit braker 101F1 tripped  statistics
      "230VAC_CB101F4Tripped" : "UDT_EventStatistic";   // Circuit braker 101F4 tripped statistics
      "230VAC_CB102F1Tripped" : "UDT_EventStatistic";   // Circuit braker 102F1 tripped statistics
      "230VAC_CB102F3Tripped" : "UDT_EventStatistic";   // Circuit braker 102F3 tripped statistics
      "230VAC_CB201F4Tripped" : "UDT_EventStatistic";   // Circuit braker 201F4 tripped statistics
      "24VDC_CB201F1Tripped" : "UDT_EventStatistic";   // Circuit braker 201F1 tripped statistics
      "24VDC_CB205F5Tripped" : "UDT_EventStatistic";   // Circuit braker 205F5 tripped statistics
      "24VDC_CB205F9Tripped" : "UDT_EventStatistic";   // Circuit braker 205F9 tripped statistics
      ScalanceSwitchStatus : "UDT_EventStatistic";   // Scalance switch status statistics
      Spare_1 : "UDT_EventStatistic";   // Spare
      Spare_2 : "UDT_EventStatistic";   // Spare
      Spare_3 : "UDT_EventStatistic";   // Spare
      PS_201T1_Tripped { S7_SetPoint := 'False'} : "UDT_EventStatistic";   // Circuit braker 201T1 tripped statistics
      "PN/PNCouplerFault" : "UDT_EventStatistic";   // PN/PN coupler fault statistics
      SingulatorCouplerFault : "UDT_EventStatistic";   // ProSoft coupler fault statistics
      ScalanceSwitchFault : "UDT_EventStatistic";   // Scalance switch fault statistics
      IOModuleCouplerFault : "UDT_EventStatistic";   // IO Module fault statistics
      RackModuleFault : "UDT_EventStatistic";   // A module fault occurred in the mainrack
   END_STRUCT;

END_TYPE

TYPE "UDT_SystemControlCommand"
TITLE = UDT_SystemControlCommand
VERSION : 0.1
//User-defined structure of system control commands.
   STRUCT
      Start { ExternalAccessible := 'False'; ExternalVisible := 'False'; ExternalWritable := 'False'} : Bool;   // Start Command from HMI
      Stop { ExternalAccessible := 'False'; ExternalVisible := 'False'; ExternalWritable := 'False'} : Bool;   // Stop command from HMI
      Reset { ExternalAccessible := 'False'; ExternalVisible := 'False'; ExternalWritable := 'False'} : Bool;   // Reset command from HMI
      ResetData { ExternalAccessible := 'False'; ExternalVisible := 'False'; ExternalWritable := 'False'} : Bool;   // Reset data command from HMI
      ResetSafety { ExternalAccessible := 'False'; ExternalVisible := 'False'; ExternalWritable := 'False'} : Bool;   // Reset safety command from HMI
      ManualMode { ExternalAccessible := 'False'; ExternalVisible := 'False'; ExternalWritable := 'False'} : Bool;   // Manual mode command from HMI
   END_STRUCT;

END_TYPE

DATA_BLOCK "DB_FIFOMedPrioMsg"
TITLE = DB_FIFO
{ S7_Optimized_Access := 'TRUE' }
AUTHOR : MHSE
FAMILY : GeneralSystemFunctions
VERSION : 3.0
NON_RETAIN
//Data block to store FIFO registers.
   VAR RETAIN
      Header { ExternalAccessible := 'False'; ExternalVisible := 'False'; ExternalWritable := 'False'; S7_SetPoint := 'False'} : "UDT_FifoHeader";   // FIFO Header
      Data { ExternalAccessible := 'False'; ExternalVisible := 'False'; ExternalWritable := 'False'; S7_SetPoint := 'False'} : Array[0..199] of "UDT_Message";   // FIFO data buffer
   END_VAR


BEGIN

END_DATA_BLOCK

DATA_BLOCK "DB_FIFORcvMsg"
TITLE = DB_FIFO
{ S7_Optimized_Access := 'TRUE' }
AUTHOR : MHSE
FAMILY : GeneralSystemFunctions
VERSION : 3.0
NON_RETAIN
//Data block to store FIFO registers.
   VAR RETAIN
      Header { ExternalAccessible := 'False'; ExternalVisible := 'False'; ExternalWritable := 'False'; S7_SetPoint := 'False'} : "UDT_FifoHeader";   // FIFO Header
      Data { ExternalAccessible := 'False'; ExternalVisible := 'False'; ExternalWritable := 'False'; S7_SetPoint := 'False'} : Array[0..199] of "UDT_Message";   // FIFO data buffer
   END_VAR


BEGIN

END_DATA_BLOCK

DATA_BLOCK "DB_Configuration"
TITLE = DB_Configuration
{ S7_Optimized_Access := 'TRUE' }
AUTHOR : MHSE
FAMILY : GeneralSystemFunctions
VERSION : 3.0
NON_RETAIN
//Data block to store configuration data.
   VAR RETAIN
      System { ExternalAccessible := 'False'; ExternalVisible := 'False'; ExternalWritable := 'False'} : Struct   // System configuration
         Connection { ExternalAccessible := 'False'; ExternalVisible := 'False'; ExternalWritable := 'False'} : "UDT_Connection";   // Connection configuration
      END_STRUCT;
   END_VAR


BEGIN
   System.Connection.ActiveEstablished := TRUE;
   System.Connection.Interface_ID := 64;
   System.Connection.ID := 16#0001;
   System.Connection.IP[1] := 192;
   System.Connection.IP[2] := 168;
   System.Connection.IP[3] := 3;
   System.Connection.IP[4] := 53;
   System.Connection.Port := 42300;
   System.Connection.ConTimeout := 5000;

END_DATA_BLOCK

DATA_BLOCK "DB_FIFOHighPrioMsg"
TITLE = DB_FIFO
{ S7_Optimized_Access := 'TRUE' }
AUTHOR : MHSE
FAMILY : GeneralSystemFunctions
VERSION : 3.0
NON_RETAIN
//Data block to store FIFO registers.
   VAR
      Header { ExternalAccessible := 'False'; ExternalVisible := 'False'; ExternalWritable := 'False'; S7_SetPoint := 'False'} : "UDT_FifoHeader";   // FIFO Header
      Data { ExternalAccessible := 'False'; ExternalVisible := 'False'; ExternalWritable := 'False'; S7_SetPoint := 'False'} : Array[0..199] of "UDT_Message";   // FIFO data buffer
   END_VAR


BEGIN

END_DATA_BLOCK

DATA_BLOCK "DB_ExternalHandshake"
TITLE = DB_ExternalHandshake
{ S7_Optimized_Access := 'TRUE' }
AUTHOR : MHSE
FAMILY : Equimpent
VERSION : 3.0
NON_RETAIN
//Data block to store external equipment handshake data.

BEGIN

END_DATA_BLOCK

DATA_BLOCK "DB_Control"
{ S7_Optimized_Access := 'TRUE' }
AUTHOR : MHSE
FAMILY : Equimpent
VERSION : 0.1
NON_RETAIN
   VAR
      System1 { ExternalAccessible := 'False'; ExternalVisible := 'False'; ExternalWritable := 'False'; S7_SetPoint := 'False'} : "UDT_EquipmentControl";
   END_VAR


BEGIN

END_DATA_BLOCK

DATA_BLOCK "DB_Communication"
TITLE = DB_Communication
{ S7_Optimized_Access := 'TRUE' }
AUTHOR : MHSE
FAMILY : Communication
VERSION : 3.0
NON_RETAIN
//Data block to store communication data.
   VAR
      BuildingMnemonic { ExternalAccessible := 'False'; ExternalVisible := 'False'; ExternalWritable := 'False'} : String[5];   // Building mnemonic
      ModuleName { ExternalAccessible := 'False'; ExternalVisible := 'False'; ExternalWritable := 'False'} : String[2];   // Module type
      DeviceNumber { ExternalAccessible := 'False'; ExternalVisible := 'False'; ExternalWritable := 'False'} : String[4];   // Device number
   END_VAR


BEGIN
   BuildingMnemonic := 'abcde';
   ModuleName := 'AB';
   DeviceNumber := 'abcd';

END_DATA_BLOCK

DATA_BLOCK "DB_WSRManager"
{ S7_Optimized_Access := 'TRUE' }
VERSION : 0.1
NON_RETAIN
   VAR
      EmptyFifoHeader { ExternalAccessible := 'False'; ExternalVisible := 'False'; ExternalWritable := 'False'; S7_SetPoint := 'False'} : "UDT_FifoHeader";
      EmptyFifoData { ExternalAccessible := 'False'; ExternalVisible := 'False'; ExternalWritable := 'False'} : Array[0..110] of Int;
      PartialFifoHeader { ExternalAccessible := 'False'; ExternalVisible := 'False'; ExternalWritable := 'False'; S7_SetPoint := 'False'} : "UDT_FifoHeader";
      PartialFifoData { ExternalAccessible := 'False'; ExternalVisible := 'False'; ExternalWritable := 'False'} : Array[0..110] of Int;
      WSR01Empty { ExternalAccessible := 'False'; ExternalVisible := 'False'; ExternalWritable := 'False'; S7_SetPoint := 'False'} : Array[0..18] of "UDT_WSRBufferState";
      WSR01Partial { ExternalAccessible := 'False'; ExternalVisible := 'False'; ExternalWritable := 'False'; S7_SetPoint := 'False'} : Array[0..18] of "UDT_WSRBufferState";
   END_VAR


BEGIN

END_DATA_BLOCK

DATA_BLOCK "DB_RATPositioning"
{ S7_Optimized_Access := 'TRUE' }
VERSION : 0.1
NON_RETAIN

BEGIN

END_DATA_BLOCK

DATA_BLOCK "DB_GOSLog"
{ S7_Optimized_Access := 'TRUE' }
VERSION : 0.1
NON_RETAIN
   VAR
      DB_GOSLog { ExternalAccessible := 'False'; ExternalVisible := 'False'; ExternalWritable := 'False'; S7_SetPoint := 'False'} : Array[0..100] of "UDT_GOSLog";
   END_VAR


BEGIN

END_DATA_BLOCK

DATA_BLOCK "DB_ExternalGIN"
{ S7_Optimized_Access := 'TRUE' }
VERSION : 0.1
NON_RETAIN
   VAR
      UnexpectedSI { ExternalAccessible := 'False'; ExternalVisible := 'False'; ExternalWritable := 'False'; S7_SetPoint := 'False'} : "UDT_GIN";
   END_VAR


BEGIN

END_DATA_BLOCK

DATA_BLOCK "DB_HMISpeed"
{ S7_Optimized_Access := 'TRUE' }
VERSION : 0.1
NON_RETAIN
   VAR
      Dummy : Int;
   END_VAR


BEGIN

END_DATA_BLOCK

DATA_BLOCK "DB_Variables"
{ S7_Optimized_Access := 'TRUE' }
VERSION : 0.1
NON_RETAIN
   VAR
      CIP_StopRequest { ExternalAccessible := 'False'; ExternalVisible := 'False'; ExternalWritable := 'False'} : Bool;   // System stop request from CIP
      ResetEnergySave { ExternalAccessible := 'False'; ExternalVisible := 'False'; ExternalWritable := 'False'} : Bool;   // When True Reset Energy Save mode
      StartToSystemControl { ExternalAccessible := 'False'; ExternalVisible := 'False'; ExternalWritable := 'False'} : Bool;   // From SSP Lamp to System Control
      ResetToSystemControl { ExternalAccessible := 'False'; ExternalVisible := 'False'; ExternalWritable := 'False'} : Bool;   // From SSP Lamp to System Control
   END_VAR


BEGIN

END_DATA_BLOCK

DATA_BLOCK "DB_FIFOLowPrioMsg"
TITLE = DB_FIFO
{ S7_Optimized_Access := 'TRUE' }
AUTHOR : MHSE
FAMILY : GeneralSystemFunctions
VERSION : 3.0
NON_RETAIN
//Data block to store FIFO registers.
   VAR RETAIN
      Header { ExternalAccessible := 'False'; ExternalVisible := 'False'; ExternalWritable := 'False'; S7_SetPoint := 'False'} : "UDT_FifoHeader";   // FIFO Header
      Data { ExternalAccessible := 'False'; ExternalVisible := 'False'; ExternalWritable := 'False'; S7_SetPoint := 'False'} : Array[0..199] of "UDT_Message";   // FIFO data buffer
   END_VAR


BEGIN

END_DATA_BLOCK

DATA_BLOCK "DB_ProgrammingError"
{ S7_Optimized_Access := 'TRUE' }
VERSION : 0.1
NON_RETAIN
   VAR
      NrOfErrors { ExternalAccessible := 'False'; ExternalVisible := 'False'; ExternalWritable := 'False'} : Int;
      BlockNr { ExternalAccessible := 'False'; ExternalVisible := 'False'; ExternalWritable := 'False'} : UInt;
      Reaction { ExternalAccessible := 'False'; ExternalVisible := 'False'; ExternalWritable := 'False'} : USInt;
      Fault_ID { ExternalAccessible := 'False'; ExternalVisible := 'False'; ExternalWritable := 'False'} : Byte;
      BlockType { ExternalAccessible := 'False'; ExternalVisible := 'False'; ExternalWritable := 'False'} : USInt;
      Area { ExternalAccessible := 'False'; ExternalVisible := 'False'; ExternalWritable := 'False'} : USInt;
      DBNr { ExternalAccessible := 'False'; ExternalVisible := 'False'; ExternalWritable := 'False'} : DB_ANY;
      Csg_OBNr { ExternalAccessible := 'False'; ExternalVisible := 'False'; ExternalWritable := 'False'} : OB_ANY;
      Csg_Prio { ExternalAccessible := 'False'; ExternalVisible := 'False'; ExternalWritable := 'False'} : USInt;
      Width { ExternalAccessible := 'False'; ExternalVisible := 'False'; ExternalWritable := 'False'} : USInt;
   END_VAR


BEGIN

END_DATA_BLOCK

DATA_BLOCK "DB_HMIStatusConfiguration"
TITLE = DB_HMIStatusConfiguration
{ S7_Optimized_Access := 'TRUE' }
AUTHOR : MHSE
VERSION : 3.0
NON_RETAIN
   VAR
      FireAlarm : Int;   // Fire alarm active
      SafetyStop : Int;   // Safety stop error status
      Error : Int;   // Error status
      Warning : Int;   // Warning status
      ManualRun : Int;   // Manual run status
      Manual : Int;   // Manual status
      Halted : Int;   // Halted status
      Dieback : Int;   // Die back status
      Stopped : Int;   // Stopped status
      Running : Int;   // Running status
      EnergySave : Int;   // Energy save status
      CommunicationError : Int;   // Communication error status
      CBError : Int;   // CB error status
      ProfinetError : Int;   // Profinet error status
      HardwareError : Int;   // Hardware error status
      VFDNotHealthy : Int;   // VFD noth healthy status
      VFDError : Int;   // VFD error status
      PECJam : Int;   // PEC jam status
      ChuteFull : Int;   // Chute full status
      EncoderError : Int;   // Encoder error status
      TrackingError : Int;   // Tracking error status
      DimensionError : Int;   // Dimension error status
      OperationalError : Int;   // Operational error status
      AutoON : Int;   // Automatic is on
      ChuteHalfFull : Int;   // Disable by operator
      DisableByManagement : Int;   // Disable by management
      GateOpen : Int;   // Manual operated gate is open
      GateClosed : Int;   // Manual operated gate is closed
      GateClosedAndNoOperatorPresent : Int;   // Manual operated gate is closed and no operator is present
      PositionChangeOngoing : Int;   // Lifting device or arm diverter changing position
      BufferMode : Int;   // BufferMode Active
      ContinuousMode : Int;   // ContinuousMode Active
      LabbelingMode : Int;   // LabbelingMode Active
   END_VAR


BEGIN
   FireAlarm := 1;
   SafetyStop := 3;
   Error := 5;
   Warning := 7;
   ManualRun := 9;
   Manual := 11;
   Halted := 13;
   Dieback := 15;
   Stopped := 17;
   Running := 19;
   EnergySave := 21;
   CommunicationError := 23;
   CBError := 25;
   ProfinetError := 27;
   HardwareError := 29;
   VFDNotHealthy := 31;
   VFDError := 33;
   PECJam := 35;
   ChuteFull := 37;
   EncoderError := 39;
   TrackingError := 41;
   DimensionError := 43;
   OperationalError := 45;
   AutoON := 47;
   ChuteHalfFull := 49;
   DisableByManagement := 51;
   GateOpen := 53;
   GateClosed := 55;
   GateClosedAndNoOperatorPresent := 57;
   PositionChangeOngoing := 59;
   BufferMode := 61;
   ContinuousMode := 63;
   LabbelingMode := 65;

END_DATA_BLOCK

DATA_BLOCK "DB_Handshake"
TITLE = DB_Handshake
{ S7_Optimized_Access := 'TRUE' }
AUTHOR : MHSE
FAMILY : Equimpent
VERSION : 3.0
NON_RETAIN
//Data block to store equipment handshake data.

BEGIN

END_DATA_BLOCK

DATA_BLOCK "DB_SafetyInterface"
{ S7_Optimized_Access := 'TRUE' }
VERSION : 0.1
NON_RETAIN
   VAR
      SafetyReset { ExternalAccessible := 'False'; ExternalVisible := 'False'; ExternalWritable := 'False'} : Bool;
   END_VAR


BEGIN

END_DATA_BLOCK

DATA_BLOCK "DB_MotorData"
{ S7_Optimized_Access := 'TRUE' }
VERSION : 0.1
NON_RETAIN

BEGIN

END_DATA_BLOCK

DATA_BLOCK "DB_VFDCommissioningControl"
{ S7_Optimized_Access := 'TRUE' }
VERSION : 0.1
NON_RETAIN
   VAR
      dummy_Start { ExternalAccessible := 'False'; ExternalVisible := 'False'; ExternalWritable := 'False'} : Bool;   // start VFD Commissioning
      dummy_GoToNextStep { ExternalAccessible := 'False'; ExternalVisible := 'False'; ExternalWritable := 'False'} : Bool;   // Trigger to move into the next step
   END_VAR


BEGIN

END_DATA_BLOCK

DATA_BLOCK "DB_HardwareOK"
{ S7_Optimized_Access := 'TRUE' }
VERSION : 0.1
NON_RETAIN
   VAR
      System { ExternalAccessible := 'False'; ExternalVisible := 'False'; ExternalWritable := 'False'} : Struct   // System status
         MCP { ExternalAccessible := 'False'; ExternalVisible := 'False'; ExternalWritable := 'False'} : Bool;   // Main Control Panel
         CPG01 { ExternalAccessible := 'False'; ExternalVisible := 'False'; ExternalWritable := 'False'} : Bool;
      END_STRUCT;
   END_VAR


BEGIN

END_DATA_BLOCK

DATA_BLOCK "DB_CommonStatus"
TITLE = DB_Status
{ S7_Optimized_Access := 'TRUE' }
AUTHOR : MHSE
FAMILY : GeneralSystemFunctions
VERSION : 3.0
NON_RETAIN
//Data block to store status data.
   VAR
      Communication : Struct   // Communication status
         TCPIPConnect : "UDT_CommonStatus";   // FB_TCPIPConnect status
      END_STRUCT;
      System : Struct   // System statuses
         System1 { S7_SetPoint := 'False'} : "UDT_CommonStatus";
         MCP { S7_SetPoint := 'False'} : "UDT_CommonStatus";
         CPG01 : "UDT_CommonStatus";
         CPG02 : "UDT_CommonStatus";
         CPG03 : "UDT_CommonStatus";
         CPG04 : "UDT_CommonStatus";
         CPG05 : "UDT_CommonStatus";
         test { S7_SetPoint := 'True'} : Int;
      END_STRUCT;
   END_VAR


BEGIN

END_DATA_BLOCK

DATA_BLOCK "DB_UnknownGINRange"
TITLE = DB_UnknownGINRange
{ S7_Optimized_Access := 'TRUE' }
AUTHOR : MHSE
FAMILY : GeneralSystemFunctions
VERSION : 3.0
NON_RETAIN
//Data block to store unknown GIN range data.
   VAR RETAIN
      UnknownGINRange { ExternalAccessible := 'False'; ExternalVisible := 'False'; ExternalWritable := 'False'; S7_SetPoint := 'False'} : "UDT_UnknownGIN";   // Unknown GIN range structure
   END_VAR


BEGIN

END_DATA_BLOCK

DATA_BLOCK "DB_Time"
TITLE = DB_Time
{ S7_Optimized_Access := 'TRUE' }
AUTHOR : MHSE
FAMILY : GeneralSystemFunctions
VERSION : 3.0
NON_RETAIN
//Data block to store date and time data.
   VAR
      ActualTimeDTL {InstructionName := 'DTL'; LibVersion := '1.0'; ExternalAccessible := 'False'; ExternalVisible := 'False'; ExternalWritable := 'False'} : DTL;   // Actual date and time in DTL
      ActualTime { ExternalAccessible := 'False'; ExternalVisible := 'False'; ExternalWritable := 'False'} : String;   // Actual date and time in String
      Timestamp { ExternalAccessible := 'False'; ExternalVisible := 'False'; ExternalWritable := 'False'} : String[17];   // Actual date and time in String
      DaylightSaving { ExternalAccessible := 'False'; ExternalVisible := 'False'; ExternalWritable := 'False'} : Int;
   END_VAR


BEGIN

END_DATA_BLOCK

DATA_BLOCK "DB_Status"
TITLE = DB_Status
{ S7_Optimized_Access := 'TRUE' }
AUTHOR : MHSE
FAMILY : GeneralSystemFunctions
VERSION : 3.0
NON_RETAIN
//Data block to store status data.
   VAR
      Communication : Struct   // Communication status
         TCPIPConnect : "UDT_TCPIPConnectStatus";   // FB_TCPIPConnect status
      END_STRUCT;
      System : Struct   // System status
         MCP { S7_SetPoint := 'False'} : "UDT_MainControlPanelStatus";   // Status of Main Control Panel
         CPG01 : "UDT_ControlPowerGroupStatus";   // Status of  Control Power Group 01
         CPG02 : "UDT_ControlPowerGroupStatus";   // Status of  Control Power Group 02
         CPG03 : "UDT_ControlPowerGroupStatus";   // Status of  Control Power Group 03
         CPG04 : "UDT_ControlPowerGroupStatus";   // Status of  Control Power Group 04
         CPG05 : "UDT_ControlPowerGroupStatus";   // Status of  Control Power Group 05
         System1 : "UDT_SystemControlStatus";
      END_STRUCT;
   END_VAR


BEGIN

END_DATA_BLOCK

DATA_BLOCK "DB_Statistics"
TITLE = DB_Statistics
{ S7_Optimized_Access := 'TRUE' }
AUTHOR : MHSE
FAMILY : GeneralSystemFunctions
VERSION : 3.0
NON_RETAIN
//Data block to store statistical data.
   VAR
      Communication : Struct   // Communication statistic
         TCPIPConnect : "UDT_TCPIPConnectStatistics";   // TCPIP Connect statistics
         TCPIPReceive : "UDT_TCPIPReceiveStatistics";   // TCPIP Receive statistics
      END_STRUCT;
      System : Struct   // System statistic
         MCP { S7_SetPoint := 'False'} : "UDT_MainControlPanelStatistics";   // Statistics of Main Control Panel
         CPG01 : "UDT_ControlPowerGroupStatistics";   // Statistics of  Control Power Group 01
         CPG02 : "UDT_ControlPowerGroupStatistics";   // Statistics of  Control Power Group 02
         CPG03 : "UDT_ControlPowerGroupStatistics";   // Statistics of  Control Power Group 03
         CPG04 : "UDT_ControlPowerGroupStatistics";   // Statistics of  Control Power Group 04
         CPG05 : "UDT_ControlPowerGroupStatistics";   // Statistics of  Control Power Group 05
         Profinet { S7_SetPoint := 'False'} : "UDT_ProfiDiagStatistics";
      END_STRUCT;
   END_VAR


BEGIN

END_DATA_BLOCK

DATA_BLOCK "DB_SoftwareVersion"
TITLE = DB_SoftwareVersion
{ S7_Optimized_Access := 'TRUE' }
AUTHOR : MHSE
FAMILY : GeneralSystemFunctions
VERSION : 3.0
NON_RETAIN
//Data block to store software version data.
   VAR
      "Version" { ExternalAccessible := 'False'; ExternalVisible := 'False'; ExternalWritable := 'False'} : String[8];   // Software version
      StandardChecksum { ExternalAccessible := 'False'; ExternalVisible := 'False'; ExternalWritable := 'False'} : Array[0..7] of Byte;   // Standard program checksum
      SafetyChecksum { ExternalAccessible := 'False'; ExternalVisible := 'False'; ExternalWritable := 'False'} : Array[0..7] of Byte;   // Safety program checksum
   END_VAR


BEGIN

END_DATA_BLOCK

DATA_BLOCK "DB_ProfinetDiagnostic"
TITLE = DB_ProfinetDiagnostic
{ S7_Optimized_Access := 'TRUE' }
AUTHOR : MHSE
FAMILY : GeneralSystemFunctions
VERSION : 3.0
NON_RETAIN
//Data block to store profinet network diagnostic data.
   VAR
      ProfinetNetworks { ExternalAccessible := 'False'; ExternalVisible := 'False'; ExternalWritable := 'False'; S7_SetPoint := 'False'} : Array[1..10] of "UDT_ProfinetNetwork";
   END_VAR


BEGIN

END_DATA_BLOCK

DATA_BLOCK "DB_PowerDistributionPanel"
TITLE = DB_PDP
{ S7_Optimized_Access := 'TRUE' }
AUTHOR : MHSE
VERSION : 3.0
NON_RETAIN
   VAR
      PDP01 { ExternalAccessible := 'False'; ExternalVisible := 'False'; ExternalWritable := 'False'; S7_SetPoint := 'False'} : "UDT_PowerDistributionPanelCBState";   // State of PDP01 Circuit Breakers
      PDP02 { ExternalAccessible := 'False'; ExternalVisible := 'False'; ExternalWritable := 'False'; S7_SetPoint := 'False'} : "UDT_PowerDistributionPanelCBState";   // State of PDP02 Circuit Breakers
      PDP03 { ExternalAccessible := 'False'; ExternalVisible := 'False'; ExternalWritable := 'False'; S7_SetPoint := 'False'} : "UDT_PowerDistributionPanelCBState";   // State of PDP03 Circuit Breakers
      PDP04 { ExternalAccessible := 'False'; ExternalVisible := 'False'; ExternalWritable := 'False'; S7_SetPoint := 'False'} : "UDT_PowerDistributionPanelCBState";   // State of PDP04 Circuit Breakers
      PDP05 { ExternalAccessible := 'False'; ExternalVisible := 'False'; ExternalWritable := 'False'; S7_SetPoint := 'False'} : "UDT_PowerDistributionPanelCBState";   // State of PDP05 Circuit Breakers
      PDP06 { ExternalAccessible := 'False'; ExternalVisible := 'False'; ExternalWritable := 'False'; S7_SetPoint := 'False'} : "UDT_PowerDistributionPanelCBState";   // State of PDP06 Circuit Breakers
      PDP07 { ExternalAccessible := 'False'; ExternalVisible := 'False'; ExternalWritable := 'False'; S7_SetPoint := 'False'} : "UDT_PowerDistributionPanelCBState";   // State of PDP07 Circuit Breakers
      PDP08 { ExternalAccessible := 'False'; ExternalVisible := 'False'; ExternalWritable := 'False'; S7_SetPoint := 'False'} : "UDT_PowerDistributionPanelCBState";   // State of PDP08 Circuit Breakers
      PDP09 { ExternalAccessible := 'False'; ExternalVisible := 'False'; ExternalWritable := 'False'; S7_SetPoint := 'False'} : "UDT_PowerDistributionPanelCBState";   // State of PDP09 Circuit Breakers
      PDP10 { ExternalAccessible := 'False'; ExternalVisible := 'False'; ExternalWritable := 'False'; S7_SetPoint := 'False'} : "UDT_PowerDistributionPanelCBState";   // State of PDP10 Circuit Breakers
   END_VAR


BEGIN

END_DATA_BLOCK

DATA_BLOCK "DB_ParametrizationErrors"
TITLE = DB_ParametrizationErrors
{ S7_Optimized_Access := 'TRUE' }
AUTHOR : MHSE
FAMILY : GeneralSystemFunctions
VERSION : 3.0
NON_RETAIN
//Data block to store parametrization errors.
   VAR
      System { ExternalAccessible := 'False'; ExternalVisible := 'False'; ExternalWritable := 'False'} : Struct
         Communication { ExternalAccessible := 'False'; ExternalVisible := 'False'; ExternalWritable := 'False'} : Struct
            TCPIPSendError { ExternalAccessible := 'False'; ExternalVisible := 'False'; ExternalWritable := 'False'} : Bool;   // TCPIP send error
            TCPIPSendWarning { ExternalAccessible := 'False'; ExternalVisible := 'False'; ExternalWritable := 'False'} : Bool;   // TCPIP send warning
            TCPIPReceiveError { ExternalAccessible := 'False'; ExternalVisible := 'False'; ExternalWritable := 'False'} : Bool;   // TCPIP receive error
            TCPIPReceiveWarning { ExternalAccessible := 'False'; ExternalVisible := 'False'; ExternalWritable := 'False'} : Bool;   // TCPIP receive warning
         END_STRUCT;
      END_STRUCT;
   END_VAR


BEGIN

END_DATA_BLOCK

DATA_BLOCK "DB_Memory"
TITLE = DB_Memory
{ S7_Optimized_Access := 'TRUE' }
AUTHOR : MHSE
VERSION : 3.0
NON_RETAIN
   VAR
      ClockByte { ExternalAccessible := 'False'; ExternalVisible := 'False'; ExternalWritable := 'False'} : Byte;   // System clock byte
      Clock_10Hz { ExternalAccessible := 'False'; ExternalVisible := 'False'; ExternalWritable := 'False'} : Bool;   // 10 Hz system clock bit
      Clock_5Hz { ExternalAccessible := 'False'; ExternalVisible := 'False'; ExternalWritable := 'False'} : Bool;   // 5 Hz system clock bit
      "Clock_2.5Hz" { ExternalAccessible := 'False'; ExternalVisible := 'False'; ExternalWritable := 'False'} : Bool;   // 2.5 Hz system clock bit
      Clock_2Hz { ExternalAccessible := 'False'; ExternalVisible := 'False'; ExternalWritable := 'False'} : Bool;   // 2 Hz system clock bit
      "Clock_1.25Hz" { ExternalAccessible := 'False'; ExternalVisible := 'False'; ExternalWritable := 'False'} : Bool;   // 1.25 Hz system clock bit
      Clock_1Hz { ExternalAccessible := 'False'; ExternalVisible := 'False'; ExternalWritable := 'False'} : Bool;   // 1 Hz system clock bit
      "Clock_0.625Hz" { ExternalAccessible := 'False'; ExternalVisible := 'False'; ExternalWritable := 'False'} : Bool;   // 0.625 Hz system clock bit
      "Clock_0.5Hz" { ExternalAccessible := 'False'; ExternalVisible := 'False'; ExternalWritable := 'False'} : Bool;   // 0.5 Hz system clock bit
      SystemByte { ExternalAccessible := 'False'; ExternalVisible := 'False'; ExternalWritable := 'False'} : Byte;   // System byte
      OSClockByte { ExternalAccessible := 'False'; ExternalVisible := 'False'; ExternalWritable := 'False'} : Byte;   // One shot of clock pulse
      "OS_0.1sec" { ExternalAccessible := 'False'; ExternalVisible := 'False'; ExternalWritable := 'False'} : Bool;   // One shot every 0.1 sec
      "OS_0.2sec" { ExternalAccessible := 'False'; ExternalVisible := 'False'; ExternalWritable := 'False'} : Bool;   // One shot every 0.2 sec
      "OS_0.4sec" { ExternalAccessible := 'False'; ExternalVisible := 'False'; ExternalWritable := 'False'} : Bool;   // One shot every 0.4 sec
      "OS_0.5sec" { ExternalAccessible := 'False'; ExternalVisible := 'False'; ExternalWritable := 'False'} : Bool;   // One shot every 0.5 sec
      "OS_0.8sec" { ExternalAccessible := 'False'; ExternalVisible := 'False'; ExternalWritable := 'False'} : Bool;   // One shot every 0.8 sec
      OS_1sec { ExternalAccessible := 'False'; ExternalVisible := 'False'; ExternalWritable := 'False'} : Bool;   // One shot every 1 sec
      "OS_1.6sec" { ExternalAccessible := 'False'; ExternalVisible := 'False'; ExternalWritable := 'False'} : Bool;   // One shot every 1.6 sec
      OS_2sec { ExternalAccessible := 'False'; ExternalVisible := 'False'; ExternalWritable := 'False'} : Bool;   // One shot every 2 sec
      PrevCycleTime { ExternalAccessible := 'False'; ExternalVisible := 'False'; ExternalWritable := 'False'} : LReal;   // Previous PLC cycle Time
      RuntimeMem { ExternalAccessible := 'False'; ExternalVisible := 'False'; ExternalWritable := 'False'} : LReal;   // Runtime memory
      FirstScan { ExternalAccessible := 'False'; ExternalVisible := 'False'; ExternalWritable := 'False'} : Bool;   // First scan bit
      DiagStatusUpdate { ExternalAccessible := 'False'; ExternalVisible := 'False'; ExternalWritable := 'False'} : Bool;   // Diagnostic status update
      AlwaysTrue { ExternalAccessible := 'False'; ExternalVisible := 'False'; ExternalWritable := 'False'} : Bool;   // Always True bit
      AlwaysFalse { ExternalAccessible := 'False'; ExternalVisible := 'False'; ExternalWritable := 'False'} : Bool;   // Always False bit
      CommissioningFalse { ExternalAccessible := 'False'; ExternalVisible := 'False'; ExternalWritable := 'False'} : Bool;   // Commissioning always false
      CommissioningTrue { ExternalAccessible := 'False'; ExternalVisible := 'False'; ExternalWritable := 'False'} : Bool;   // Commissioning always true
      ReconnectCommand { ExternalAccessible := 'False'; ExternalVisible := 'False'; ExternalWritable := 'False'} : Bool;   // Reconnect command
      ScanMainRack { ExternalAccessible := 'False'; ExternalVisible := 'False'; ExternalWritable := 'False'} : Bool;   // Trigger to check main rack confiuration
      ScanProfinet { ExternalAccessible := 'False'; ExternalVisible := 'False'; ExternalWritable := 'False'} : Bool;   // Scan profinet bit
      Simulation { ExternalAccessible := 'False'; ExternalVisible := 'False'; ExternalWritable := 'False'} : Bool;   // Simulation
      PN1OK { ExternalAccessible := 'False'; ExternalVisible := 'False'; ExternalWritable := 'False'} : Bool;   // Profinet ok
      "Local~PROFINET_IO-System" { ExternalAccessible := 'False'; ExternalVisible := 'False'; ExternalWritable := 'False'} : HW_ANY;   // HW Intentifier of PN-IO System
      "Local~PROFINET_IO-System_1" { ExternalAccessible := 'False'; ExternalVisible := 'False'; ExternalWritable := 'False'} : HW_ANY;   // HW Intentifier of PN-IOSystem 1
      "Local~PROFINET_IO-System_2" { ExternalAccessible := 'False'; ExternalVisible := 'False'; ExternalWritable := 'False'} : HW_ANY;   // HW Intentifier of PN-IOSystem 2
      "Local~PROFINET_IO-System_3" { ExternalAccessible := 'False'; ExternalVisible := 'False'; ExternalWritable := 'False'} : HW_ANY;   // HW Intentifier of PN-IOSystem 3
      "Local~PROFINET_IO-System_4" { ExternalAccessible := 'False'; ExternalVisible := 'False'; ExternalWritable := 'False'} : HW_ANY;   // HW Intentifier of PN-IOSystem 4
      "Local~PROFINET_IO-System_5" { ExternalAccessible := 'False'; ExternalVisible := 'False'; ExternalWritable := 'False'} : HW_ANY;   // HW Intentifier of PN-IOSystem 5
      "Local~PROFINET_IO-System_6" { ExternalAccessible := 'False'; ExternalVisible := 'False'; ExternalWritable := 'False'} : HW_ANY;   // HW Intentifier of PN-IOSystem 6
      "Local~PROFINET_IO-System_7" { ExternalAccessible := 'False'; ExternalVisible := 'False'; ExternalWritable := 'False'} : HW_ANY;   // HW Intentifier of PN-IOSystem 7
      "Local~PROFINET_IO-System_8" { ExternalAccessible := 'False'; ExternalVisible := 'False'; ExternalWritable := 'False'} : HW_ANY;   // HW Intentifier of PN-IOSystem 8
      "Local~PROFINET_IO-System_9" { ExternalAccessible := 'False'; ExternalVisible := 'False'; ExternalWritable := 'False'} : HW_ANY;   // HW Intentifier of PN-IOSystem 9
   END_VAR


BEGIN

END_DATA_BLOCK

DATA_BLOCK "DB_Interface"
TITLE = DB_Interface
{ S7_Optimized_Access := 'TRUE' }
AUTHOR : MHSE
FAMILY : Equimpent
VERSION : 3.0
NON_RETAIN
//Data block to store equipment interface data.

BEGIN

END_DATA_BLOCK

DATA_BLOCK "DB_FIFOLostGIN"
TITLE = DB_FIFO
{ S7_Optimized_Access := 'TRUE' }
AUTHOR : MHSE
FAMILY : GeneralSystemFunctions
VERSION : 3.0
NON_RETAIN
//Data block to store FIFO registers.
   VAR RETAIN
      Header { ExternalAccessible := 'False'; ExternalVisible := 'False'; ExternalWritable := 'False'; S7_SetPoint := 'False'} : "UDT_FifoHeader";   // FIFO Header
      Data { ExternalAccessible := 'False'; ExternalVisible := 'False'; ExternalWritable := 'False'} : Array[0..199] of Int;   // FIFO data buffer
   END_VAR
   VAR
      Header_1 { ExternalAccessible := 'False'; ExternalVisible := 'False'; ExternalWritable := 'False'; S7_SetPoint := 'False'} : "UDT_FifoHeader";
      Data_1 { ExternalAccessible := 'False'; ExternalVisible := 'False'; ExternalWritable := 'False'} : Array[0..199] of Int;
      Header_2 { ExternalAccessible := 'False'; ExternalVisible := 'False'; ExternalWritable := 'False'; S7_SetPoint := 'False'} : "UDT_FifoHeader";
      Data_2 { ExternalAccessible := 'False'; ExternalVisible := 'False'; ExternalWritable := 'False'} : Array[0..199] of Int;
      Header_3 { ExternalAccessible := 'False'; ExternalVisible := 'False'; ExternalWritable := 'False'; S7_SetPoint := 'False'} : "UDT_FifoHeader";
      Data_3 { ExternalAccessible := 'False'; ExternalVisible := 'False'; ExternalWritable := 'False'} : Array[0..199] of Int;
      Header_4 { ExternalAccessible := 'False'; ExternalVisible := 'False'; ExternalWritable := 'False'; S7_SetPoint := 'False'} : "UDT_FifoHeader";
      Data_4 { ExternalAccessible := 'False'; ExternalVisible := 'False'; ExternalWritable := 'False'} : Array[0..199] of Int;
      Header_5 { ExternalAccessible := 'False'; ExternalVisible := 'False'; ExternalWritable := 'False'; S7_SetPoint := 'False'} : "UDT_FifoHeader";
      Data_5 { ExternalAccessible := 'False'; ExternalVisible := 'False'; ExternalWritable := 'False'} : Array[0..199] of Int;
      Header_6 { ExternalAccessible := 'False'; ExternalVisible := 'False'; ExternalWritable := 'False'; S7_SetPoint := 'False'} : "UDT_FifoHeader";
      Data_6 { ExternalAccessible := 'False'; ExternalVisible := 'False'; ExternalWritable := 'False'} : Array[0..199] of Int;
   END_VAR


BEGIN

END_DATA_BLOCK

DATA_BLOCK "DB_HMICommands"
TITLE = DB_HMICommands
{ S7_Optimized_Access := 'TRUE' }
AUTHOR : MHSE
FAMILY : Equimpent
VERSION : 3.0
NON_RETAIN
//Data block to store HMI commands.
   VAR
      System1 { S7_SetPoint := 'False'} : "UDT_SystemControlCommand";
   END_VAR


BEGIN

END_DATA_BLOCK

DATA_BLOCK "DB_GIN"
TITLE = DB_GIN
{ S7_Optimized_Access := 'TRUE' }
AUTHOR : MHSE
FAMILY : GeneralSystemFunctions
VERSION : 3.0
NON_RETAIN
//Data block to store parcels informations.
   VAR
      GIN { ExternalAccessible := 'False'; ExternalVisible := 'False'; ExternalWritable := 'False'; S7_SetPoint := 'False'} : Array[1..1] of "UDT_GIN";   // GIN informations - for project remove unneeded customers and extend array bound range to 9999
   END_VAR


BEGIN

END_DATA_BLOCK

DATA_BLOCK "DB_GINDefault"
{ S7_Optimized_Access := 'TRUE' }
VERSION : 0.1
NON_RETAIN
   VAR
      GIN { ExternalAccessible := 'False'; ExternalVisible := 'False'; ExternalWritable := 'False'; S7_SetPoint := 'False'} : Array[1..20] of "UDT_GIN";   // GIN informations
   END_VAR


BEGIN

END_DATA_BLOCK

